// --------------------------------------------Reworked FB from Jensen Mechatronics--------------------------------------------

FUNCTION_BLOCK FB_TcJoy IMPLEMENTS I_HMI;
VAR_INPUT
    bEnable : BOOL :=TRUE;
END_VAR
VAR_OUTPUT    
    
 // Xbox controller outputs
 stJoystickOut   : ST_Joystick_Out;
 
END_VAR
VAR
	// From VB App To PLC
	bHeartBeatToggle : BOOL;  // From VB App
	iADSWatchdogMS : DINT;    // If Rate is > this, all outputs go to 0.
	iADSWatchdogDeadDurationMS : DINT;    // If watchdog trips, outputs go to 0 for this long.
	bWatchdogFailureActive			: BOOL;
	bControllerInputsMustBeReleased  : BOOL;  // Are controller inputs holding us in latency lock down?
	// From PLC To VB (Status)
	iUpdateRateMS : DINT;    // Rate in MS between heartbeat changes detected.
	
	// Internal Use Only
	HeartBeatChanged_RTRIG : R_TRIG;
	bHeartBeatToggle_Last : BOOL;
	UpdateRate_TMR : TON;
	
	LatencyWatchdog_TMR : TON; // Watch for missing ADS and kill joy output for a while.
	LatencyWatchdogDeadDuration_TMR : TON; // Watchdog will kill the outputs for this long...
	
	iScanCount: DINT; // Scan counter for VB Status.
	
	bControllerConnected : BOOL;  // Is there a controller connected?
    
    bIsActive : BOOL;  // Are we running?
    
	// Controller Outputs for use in programs:
	Start_Button : BOOL; 
	Back_Button : BOOL;
	A_Button : BOOL;
	B_Button : BOOL;
	X_Button : BOOL;
	Y_Button : BOOL;
	LeftShoulder_Button : BOOL;
	RightShoulder_Button : BOOL;
	LeftStick_Button : BOOL;
	RightStick_Button : BOOL;
	DPad_Up_Button : BOOL;
	DPad_Left_Button : BOOL;
	DPad_Right_Button : BOOL;
	DPad_Down_Button : BOOL;
	iLeftStick_X_Axis : DINT;
	iLeftStick_Y_Axis : DINT;
	iRightStick_X_Axis : DINT;
	iRightStick_Y_Axis : DINT;
	iLeftTrigger_Axis : DINT;
	iRightTrigger_Axis  : DINT;
	sBatteryInfo		: STRING;
    
    // Jog Mode Enumeration
    nJogSelectInteger   : INT;
    eJogSelectMode      : E_JogMode;
    trigJogIncrement     : R_TRIG;
    trigJogDecrement     : R_TRIG;
 
    fbXJogScaling       : FB_CTRL_SCALE;
    stXParams           : ST_CTRL_SCALE_PARAMS;   
    fbYJogScaling       : FB_CTRL_SCALE;
    stYParams           : ST_CTRL_SCALE_PARAMS;
    fbZJogScaling       : FB_CTRL_SCALE;
    stZParams           : ST_CTRL_SCALE_PARAMS;
    fXVelocityScaled    : REAL;    
    fYVelocityScaled    : REAL;
    fZVelocityScaled    : REAL;
    bYJogPositive   : BOOL;
    bYJogNegative   : BOOL;
    bXJogPositive   : BOOL;
    bXJogNegative   : BOOL;
    bZJogPositive   : BOOL;
    bZJogNegative   : BOOL;
	
END_VAR

M_HMI_In();
M_HMI_Out();
M_XAxisControl();
M_YAxisControl();
M_ZAxisControl();
M_JogMode();
M_AxisScalingParameters();
M_Outputs();


iScanCount := iScanCount+1;

UpdateRate_TMR(PT:=T#999M);

HeartBeatChanged_RTRIG(clk := bHeartBeatToggle <> bHeartBeatToggle_Last);

// VB "Just" changed heartbeat.
IF HeartBeatChanged_RTRIG.Q THEN
	bHeartBeatToggle_Last := bHeartBeatToggle;
	iUpdateRateMS := TIME_TO_DINT(UpdateRate_TMR.ET); // Grab Elapsed Time
	UpdateRate_TMR(IN:=FALSE); // Reset Timer
	UpdateRate_TMR(IN:=TRUE); // Reset Timer
END_IF

LatencyWatchdog_TMR(IN:=bHeartBeatToggle, PT:=DINT_TO_TIME(iADSWatchdogMS));

// AHH Latency Elapsed!
IF LatencyWatchdog_TMR.Q THEN
	bWatchdogFailureActive := TRUE;
	bControllerConnected := FALSE;
END_IF

//Force User to release all buttons/sticks on controller before allowing outputs again.
IF bWatchdogFailureActive AND (Start_Button OR 
	Back_Button OR 
	A_Button OR 
	B_Button OR 
	X_Button OR 
	Y_Button OR 
	LeftShoulder_Button OR 
	RightShoulder_Button OR 
	LeftStick_Button OR
	RightStick_Button OR
	DPad_Up_Button OR 
	DPad_Left_Button OR 
	DPad_Right_Button OR 
	DPad_Down_Button OR 
	iLeftStick_X_Axis <> 0 OR
	iLeftStick_Y_Axis <> 0 OR
	iRightStick_X_Axis <> 0 OR
	iRightStick_Y_Axis <> 0 OR
	iLeftTrigger_Axis <> 0 OR
	iRightTrigger_Axis <> 0)	THEN
		bControllerInputsMustBeReleased := TRUE;
ELSE
		bControllerInputsMustBeReleased := FALSE;
END_IF

LatencyWatchdogDeadDuration_TMR(IN:=bWatchdogFailureActive AND NOT bControllerInputsMustBeReleased AND bControllerConnected, PT:=DINT_TO_TIME(iADSWatchdogDeadDurationMS));

// ReEnable after setting duration expires
IF LatencyWatchdogDeadDuration_TMR.Q THEN
	bWatchdogFailureActive := FALSE;
END_IF

// Null the outputs on WD Active so we don't jog into a wall if we lose connection.
IF (bWatchdogFailureActive OR NOT bControllerConnected OR bControllerInputsMustBeReleased) THEN
		// Null all outputs now.
		Start_Button := FALSE; 
		Back_Button := FALSE; 
		A_Button := FALSE; 
		B_Button := FALSE; 
		X_Button := FALSE; 
		Y_Button := FALSE; 
		LeftShoulder_Button := FALSE; 
		RightShoulder_Button := FALSE; 
		LeftStick_Button := FALSE; 
		RightStick_Button := FALSE; 
		DPad_Up_Button := FALSE; 
		DPad_Left_Button := FALSE; 
		DPad_Right_Button := FALSE; 
		DPad_Down_Button := FALSE; 
		iLeftStick_X_Axis := 0;
		iLeftStick_Y_Axis := 0;
		iRightStick_X_Axis := 0;
		iRightStick_Y_Axis := 0;
		iLeftTrigger_Axis := 0;
		iRightTrigger_Axis := 0;
		sBatteryInfo		:= 'Unkn';
		
		UpdateRate_TMR(IN:=FALSE); // Reset Rate Timer
ELSE
	; // All is well, VB will update our values constantly.
END_IF

bIsActive := NOT bWatchdogFailureActive AND bControllerConnected AND NOT bControllerInputsMustBeReleased;

METHOD M_AxisScalingParameters : BOOL
VAR_INPUT
END_VAR
stXParams.fInMax := 32767;
stXParams.fInMin := 0;
stXParams.fOutMax := 250.0;
stXParams.fOutMin    := 0.0;
stXParams.tCtrlCycleTime := T#100MS;
stXParams.tTaskCycleTime := T#2MS;

stYParams.fInMax := 32767;
stYParams.fInMin := 0;
stYParams.fOutMax := 245.0;
stYParams.fOutMin    := 0.0;
stYParams.tCtrlCycleTime := T#100MS;
stYParams.tTaskCycleTime := T#2MS;

stZParams.fInMax := 32767;
stZParams.fInMin := 0;
stZParams.fOutMax := 100.0;
stZParams.fOutMin    := 0.0;
stZParams.tCtrlCycleTime := T#100MS;
stZParams.tTaskCycleTime := T#2MS;
END_METHOD

METHOD M_Enable : BOOL
VAR_INPUT
END_VAR
//bEnable := ;
END_METHOD

{warning 'add method implementation '}
METHOD M_HMI_In : BOOL
//stHMI.bEnableJoystickControls
END_METHOD

{warning 'add method implementation '}
METHOD M_HMI_Out : BOOL
//stHMIOut.bXButtonPressed etc.....
END_METHOD

METHOD M_Inputs : BOOL
VAR_INPUT
END_VAR
// Make external jog controller assignments here, to internal variables for jog control

//Xbox controller mapping

//PS5 controller mapping

//Keyboard mapping

//etc...


// TcJoy inputs should be buffered here, not directly linked to variables inside the FB
END_METHOD

METHOD M_JogMode : BOOL
VAR_INPUT
END_VAR
trigJogIncrement(CLK:= RightShoulder_Button);
trigJogDecrement(CLK:= LeftShoulder_Button);


IF trigJogIncrement.Q AND nJogSelectInteger <=2 THEN    

    nJogSelectInteger := nJogSelectInteger +1;
    
ELSIF trigJogDecrement.Q AND nJogSelectInteger >=1 THEN
    nJogSelectInteger := nJogSelectInteger - 1;
    
ELSIF trigJogIncrement.Q AND nJogSelectInteger >= 3 THEN
    nJogSelectInteger :=0;
 
ELSIF trigJogDecrement.Q AND nJogSelectInteger <= 1 THEN
    nJogSelectInteger := 3;   
END_IF



CASE nJogSelectInteger  OF
    
    0:
        eJogSelectMode := MC_JOGMODE_STANDARD_SLOW;
    1:
        eJogSelectMode := MC_JOGMODE_STANDARD_FAST;
    2:
        eJogSelectMode := MC_JOGMODE_CONTINOUS;
    3:
        eJogSelectMode := MC_JOGMODE_INCHING;
    
END_CASE
END_METHOD

METHOD M_Outputs : BOOL
VAR_INPUT
END_VAR
// change this so we don't output all the keystroke/button commands, only output functions relating to MC jog using a controller. Velocity, position, jog mode, etc....
// all mapping should be handled internally in this function block




IF bEnable THEN

stJoystickOut.Start_Button := Start_Button;
stJoystickOut.Back_Button := Back_Button;
stJoystickOut.A_Button := A_Button;
stJoystickOut.B_Button := B_Button;
stJoystickOut.X_Button := X_Button;
stJoystickOut.Y_Button := Y_Button;
stJoystickOut.LeftShoulder_Button := LeftShoulder_Button; 
stJoystickOut.RightShoulder_Button := RightShoulder_Button;
stJoystickOut.LeftStick_Button := LeftStick_Button;
stJoystickOut.RightStick_Button := RightStick_Button; 
stJoystickOut.DPad_Up_Button := DPad_Up_Button;
stJoystickOut.DPad_Left_Button := DPad_Left_Button;
stJoystickOut.DPad_Right_Button := DPad_Right_Button; 
stJoystickOut.DPad_Down_Button := DPad_Down_Button;
stJoystickOut.iLeftStick_X_Axis := iLeftStick_X_Axis; 
stJoystickOut.iLeftStick_Y_Axis := iLeftStick_Y_Axis; 
stJoystickOut.iRightStick_X_Axis := iRightStick_X_Axis;
stJoystickOut.iRightStick_Y_Axis := iRightStick_Y_Axis;
stJoystickOut.iLeftTrigger_Axis := iLeftTrigger_Axis; 
stJoystickOut.iRightTrigger_Axis := iRightTrigger_Axis;


// Output buffering to MC Jog relevant functions

stJoystickOut.eJogMode      := eJogSelectMode;
stJoystickOut.bJogEnable    := (iLeftTrigger_Axis >= 230);
stJoystickOut.fXJogVelocity := fXVelocityScaled;
stJoystickOut.fYJogVelocity := fYVelocityScaled;
stJoystickOut.fZJogVelocity := fZVelocityScaled;

stJoystickOut.bXJogNegative := bXJogNegative;
stJoystickOut.bXJogPositive := bXJogPositive;

stJoystickOut.bYJogNegative := bYJogNegative;
stJoystickOut.bYJogPositive := bYJogPositive;

stJoystickOut.bZJogNegative := bZJogNegative;
stJoystickOut.bZJogPositive := bZJogPositive;

END_IF
END_METHOD

METHOD M_XAxisControl : BOOL
VAR_INPUT
END_VAR
fbXJogScaling(fIn := ABS(iLeftStick_X_Axis),
              fOut => fXVelocityScaled,
              stParams := stXParams); 
              
IF iLeftStick_X_Axis > 0 THEN
    bXJogPositive := TRUE;
ELSIF iLeftStick_X_Axis < 0 THEN
    bXJogNegative := TRUE;
ELSE
    bXJogPositive := FALSE;
    bXJogNegative := FALSE;
END_IF
END_METHOD

METHOD M_YAxisControl : BOOL
VAR_INPUT
END_VAR
fbYJogScaling(fIn := ABS(iLeftStick_Y_Axis),
              fOut => fYVelocityScaled,
              stParams := stYParams); 
              
IF iLeftStick_Y_Axis > 0 THEN
    bYJogPositive := TRUE;
ELSIF iLeftStick_Y_Axis < 0 THEN
    bYJogNegative := TRUE;
ELSE
    bYJogPositive := FALSE;
    bYJogNegative := FALSE;
END_IF
END_METHOD

METHOD M_ZAxisControl : BOOL
VAR_INPUT
END_VAR
fbZJogScaling(fIn := ABS(iRightStick_Y_Axis),
              fOut => fZVelocityScaled,
              stParams := stZParams); 
              
IF iRightStick_Y_Axis > 0 THEN
    bZJogPositive := TRUE;
ELSIF iRightStick_Y_Axis < 0 THEN
    bZJogNegative := TRUE;
ELSE
    bZJogPositive := FALSE;
    bZJogNegative := FALSE;
END_IF
END_METHOD

END_FUNCTION_BLOCK

(* stored: Version 1.1.0.1, ProductVersion 3.1.4024.11
   POU FB_TcJoy: Id {9129424f-01bc-4dfe-bce8-563189fd07db}, SpecialFunc None
   Method M_AxisScalingParameters: Id {66fc3595-2914-4900-ab15-4f39c46e81f7}
   Method M_Enable: Id {e11dbd2e-ef5b-4a80-9e37-8e9f91c38bb3}
   Method M_HMI_In: Id {0ac16883-cc0f-4b0c-9ee6-02fca7adae52}
   Method M_HMI_Out: Id {4f9129a5-2462-4ef0-8b5e-630c46ab5da3}
   Method M_Inputs: Id {44d78638-62b6-423f-a474-bf533c11d11f}
   Method M_JogMode: Id {5a525eec-016c-4cc3-9a10-42bf3e7ac809}
   Method M_Outputs: Id {f42027ab-888a-4ef2-9c42-f5eaa58e8da6}
   Method M_XAxisControl: Id {7795cb23-c6b0-45e0-b1c0-549e4a1f4ffd}
   Method M_YAxisControl: Id {96ee5d9c-40f3-4c29-bff8-bf645f9daff8}
   Method M_ZAxisControl: Id {5c308bf8-28c3-4f20-8740-ca1b719a4d46} *)
